KUKA KRL program: STOP_MAIN.src, STOP_MAIN.dat

--- STOP_MAIN.src ---
&ACCESS RVO
&REL 2
DEF  STOP_MAIN ( )
;FOLD INI;%{PE}
  ;FOLD BASISTECH INI
     IF NOT $ON_PATH THEN
    GLOBAL INTERRUPT DECL 3 WHEN $STOPMESS==TRUE DO IR_STOPM ( )
    INTERRUPT ON 3
    BAS (#INITMOV,0 )
    ENDIF
  ;ENDFOLD (BASISTECH INI)
  ;FOLD USER INI
    ;Make your modifications her

  ;ENDFOLD (USER INI)
;ENDFOLD (INI)

BRAKE
$OUT[8]=TRUE
WAIT SEC 2
WAIT FOR ( $IN[7] OR PyACK)
PyACK = FALSE
PULSE ( $OUT[7], true, 0.5 )
WAIT FOR NOT $IN[8]
$OUT[8]=FALSE
END

--- STOP_MAIN.dat ---
&ACCESS RVO
&REL 2
DEFDAT STOP_MAIN
;FOLD EXTERNAL DECLARATIONS;%{PE}%MKUKATPBASIS,%CEXT,%VCOMMON,%P
;FOLD BASISTECH EXT;%{PE}%MKUKATPBASIS,%CEXT,%VEXT,%P
EXT  BAS (BAS_COMMAND  :IN,REAL  :IN )
DECL INT SUCCESS
;ENDFOLD (BASISTECH EXT)
;FOLD USER EXT;%{E}%MKUKATPUSER,%CEXT,%VEXT,%P
;Make your modifications here

;ENDFOLD (USER EXT)
;ENDFOLD (EXTERNAL DECLARATIONS)
ENDDAT
